FUNCTION_BLOCK FB_RecipeBuilderFlaps EXTENDS FB_RecipeBase

METHOD Build : BOOL
VAR_INST
    TotalY          : REAL;
    TotalX          : REAL;
    ShorterY        : REAL;
    ShorterX        : REAL;
    
    // Zmienna lokalna, dopóki nie dodasz jej do ST_RecipeBuilder_Config
    CuttingOverpass : REAL := 20.0; 
END_VAR
TotalY   := _Config.PanelFrontLength + 2 * _Config.PanelHeight;
TotalX   := _Config.PanelFrontWidht  + 2 * _Config.PanelHeight; // Uwaga na literówkę 'Widht' w strukturze!
ShorterY := TotalY - _Config.PanelHeight;
ShorterX := TotalX - _Config.PanelHeight;


// ------------------------------------
// 1. Segregracja frezowania (Grooving)
// ------------------------------------
_SegmentsToGroove := 4;

_SegmentsGroove[1].Start.X := TotalX;
_SegmentsGroove[1].Stop.X  := 0;
_SegmentsGroove[1].Start.Y := ShorterY;
_SegmentsGroove[1].Stop.Y  := ShorterY;

_SegmentsGroove[2].Start.X := TotalX;
_SegmentsGroove[2].Stop.X  := 0; 
_SegmentsGroove[2].Start.Y := _Config.PanelHeight;
_SegmentsGroove[2].Stop.Y  := _Config.PanelHeight;

_SegmentsGroove[3].Start.X := ShorterX;
_SegmentsGroove[3].Stop.X  := ShorterX;
_SegmentsGroove[3].Start.Y := TotalY;
_SegmentsGroove[3].Stop.Y  := 0;

_SegmentsGroove[4].Start.Y := TotalY;
_SegmentsGroove[4].Stop.Y  := 0;
_SegmentsGroove[4].Start.X := _Config.PanelHeight;
_SegmentsGroove[4].Stop.X  := _Config.PanelHeight;

// ------------------------------------
// 2. Cięcie w osi X (Cut X)
// ------------------------------------
_SegmentsToCutX := 6;

// Short Box Segments
_SegmentsCutX[1].Start.X := TotalX + CuttingOverpass;
_SegmentsCutX[1].Stop.X  := ShorterX;
_SegmentsCutX[1].Start.Y := ShorterY;
_SegmentsCutX[1].Stop.Y  := ShorterY;

_SegmentsCutX[2].Start.X := _Config.PanelHeight;
_SegmentsCutX[2].Stop.X  := -CuttingOverpass;
_SegmentsCutX[2].Start.Y := ShorterY;
_SegmentsCutX[2].Stop.Y  := ShorterY;

_SegmentsCutX[3].Start.X := TotalX + CuttingOverpass;
_SegmentsCutX[3].Stop.X  := ShorterX;
_SegmentsCutX[3].Start.Y := _Config.PanelHeight;
_SegmentsCutX[3].Stop.Y  := _Config.PanelHeight;

_SegmentsCutX[4].Start.X := _Config.PanelHeight;
_SegmentsCutX[4].Stop.X  := -CuttingOverpass;
_SegmentsCutX[4].Start.Y := _Config.PanelHeight;
_SegmentsCutX[4].Stop.Y  := _Config.PanelHeight;

// Panel Dimensions Shorter Flaps
_SegmentsCutX[5].Start.X := TotalX + CuttingOverpass;
_SegmentsCutX[5].Stop.X  := -CuttingOverpass;
_SegmentsCutX[5].Start.Y := TotalY - _Config.RailHeightCorrection;
_SegmentsCutX[5].Stop.Y  := TotalY - _Config.RailHeightCorrection;

_SegmentsCutX[6].Start.X := TotalX + CuttingOverpass;
_SegmentsCutX[6].Stop.X  := -CuttingOverpass;
_SegmentsCutX[6].Start.Y := _Config.RailHeightCorrection;
_SegmentsCutX[6].Stop.Y  := _Config.RailHeightCorrection;

// ------------------------------------
// 3. Cięcie w osi Y (Cut Y)
// ------------------------------------
_SegmentsToCutY := 6;

// Short Box Segments
_SegmentsCutY[1].Start.X := ShorterX;
_SegmentsCutY[1].Stop.X  := ShorterX;
_SegmentsCutY[1].Start.Y := TotalY + CuttingOverpass;
_SegmentsCutY[1].Stop.Y  := ShorterY;

_SegmentsCutY[2].Start.X := _Config.PanelHeight;
_SegmentsCutY[2].Stop.X  := _Config.PanelHeight;
_SegmentsCutY[2].Start.Y := TotalY + CuttingOverpass;
_SegmentsCutY[2].Stop.Y  := ShorterY;

_SegmentsCutY[3].Start.X := ShorterX;
_SegmentsCutY[3].Stop.X  := ShorterX;
_SegmentsCutY[3].Start.Y := _Config.PanelHeight;
_SegmentsCutY[3].Stop.Y  := -CuttingOverpass;

_SegmentsCutY[4].Start.X := _Config.PanelHeight;
_SegmentsCutY[4].Stop.X  := _Config.PanelHeight;
_SegmentsCutY[4].Start.Y := _Config.PanelHeight;
_SegmentsCutY[4].Stop.Y  := -CuttingOverpass;

// Panel Dimensions
_SegmentsCutY[5].Start.X := TotalX;
_SegmentsCutY[5].Stop.X  := TotalX;
_SegmentsCutY[5].Start.Y := TotalY + CuttingOverpass;
_SegmentsCutY[5].Stop.Y  := -CuttingOverpass;

_SegmentsCutY[6].Start.X := 0;
_SegmentsCutY[6].Stop.X  := 0;
_SegmentsCutY[6].Start.Y := TotalY + CuttingOverpass;
_SegmentsCutY[6].Stop.Y  := -CuttingOverpass;


Build := TRUE;
END_METHOD

END_FUNCTION_BLOCK

(* stored: Version 1.1.0.1, ProductVersion 3.1.4024.15
   POU FB_RecipeBuilderFlaps: Id {1389b747-8c88-4122-8f76-112cbf46c424}, SpecialFunc None
   Method Build: Id {a7636aac-6540-4877-9111-d7366342a8fe} *)
